VAR_GLOBAL
	TestSuite : FB_TestSuite;
END_VAR

(* stored: Version 1.1.0.1
   GVL TestSuite: Id {65860d76-d62d-4014-99f3-e31b2a55eaef} *)
